TYPE ST_Homing :
STRUCT
	Mode		: SINT;
	FirstSpd		: UDINT;
	SecSpd		: UDINT;
	AccSpd		: UDINT;
END_STRUCT
END_TYPE

(* stored: Version 1.1.0.1, ProductVersion 3.1.4024.9
   DUT ST_Homing: Id {9d17cf02-bf85-4a9f-bac5-ad92391fde87} *)
